TYPE (* A Template for a Data Type *)
  (* Version 1.0, 2026-04-14, Zijun Tang *)
  PACKAGE eclipse4diac::io::ethercat;
  ECModuleConfig : STRUCT
    ModuleIdent : UDINT;
    Slot : UINT;
  END_STRUCT;
END_TYPE
